FUNCTION_BLOCK TcoTixonPickVibroSeparatorTask EXTENDS TcoTixonFeedingTask
VAR_IN_OUT
	inoConfig 	: TcoTixonPickVibro_Config_v_1_x_x;
   	inoControl 	: TcoTixonPickVibro_Control_v_1_x_x;
	inoStatus 	: TcoTixonPickVibro_Status_v_1_x_x;
END_VAR
VAR
	_componentReady: BOOL;
END_VAR

IF Execute() THEN
	 
  	IF _progress = 0 THEN
		IF NOT __ISVALIDREF(inoControl) THEN
			_varInfo :=__VARINFO(inoControl);
			Messenger.Programming(_sb.Clear().Append('<#Invalid reference: #>').Append(_varInfo.Symbol).ToString()).Pin();
		ELSIF NOT __ISVALIDREF(inoConfig) THEN                                                  
			_varInfo :=__VARINFO(inoConfig);                                                    
			Messenger.Programming(_sb.Clear().Append('<#Invalid reference: #>').Append(_varInfo.Symbol).ToString()).Pin();
		ELSIF NOT __ISVALIDREF(inoStatus) THEN                                                  
			_varInfo :=__VARINFO(inoStatus);                                                    
			Messenger.Programming(_sb.Clear().Append('<#Invalid reference: #>').Append(_varInfo.Symbol).ToString()).Pin();
		ELSIF NOT inoStatus.ControllerInAuto THEN                                                  
			_varInfo :=__VARINFO(inoStatus.ControllerInAuto);                                                                                              
			Messenger.Warning(_sb.Clear().Append('<#Tixon control system not in auto #>').Append(_varInfo.Symbol).ToString());
		ELSE

			_progress := _progress + 1;

		END_IF

	END_IF
	IF _progress = 1 THEN
		inoControl.SepareComponent:=FALSE;
		_varInfo :=__VARINFO( inoStatus.SeparatorHomePos);                                                
		THIS^.Messenger.OnCondition(_infoTimer.Q AND NOT inoStatus.SeparatorHomePos).Warning(_sb.Clear().Append('<#Waiting for #>').Append(_varInfo.Symbol).ToString());
		IF  inoStatus.SeparatorHomePos THEN
			_progress := _progress + 1;
			_timer(In:=FALSE);
		END_IF;
	END_IF;
	
	
	IF _progress = 2 THEN	
		Messenger.Debug('<#Waiting for component in  separator#>');
		_timer(IN:=inoStatus.SeparatorPresent,Pt:=inoConfig.TimeToComponentInSeparator);
		IF _timer.Q THEN
			_progress := _progress + 1;
			_timer(In:=FALSE);
		END_IF
	END_IF;
	
	IF _progress = 3 THEN	
		inoControl.SepareComponent:=TRUE;
		Messenger.Debug('<#Waiting for component out of  separator#>');
		_timer(IN:=inoStatus.SeparatorPresent,Pt:=inoConfig.TimeToComponentOutSeparator);
		IF inoStatus.SeparatorPresent THEN
			_progress := _progress + 1;
			_timer(In:=FALSE);
		ELSIF _timer.Q THEN
			_progress := 1;
			_timer(In:=FALSE);
		END_IF
	END_IF;
	
	IF _progress = 4 THEN	
		_componentReady:=TRUE;
		THIS^.DoneWhen(TRUE);
	END_IF;		

   
    CallTimers(TRUE);
	
	THIS^.ThrowWhen(_errorTimer.Q );
	
END_IF

inoStatus.ComponentReady:=_componentReady;

IF  THIS^.Error AND NOT _errorMessage.Pinned THEN
	THIS^.Restore();
END_IF

PROPERTY PUBLIC ComponentReady : bool
GET
ComponentReady:=_componentReady;
END_GET
END_PROPERTY

(*~
	<docu>
		<summary>
			Executes when task is aborted.
		</summary>			
	</docu>	
~*)
METHOD PROTECTED OnAbort
IF  __ISVALIDREF(inoStatus) THEN   THIS^.inoStatus.ActionDescription := '<#Separator task  was aborted.#>'; END_IF;
END_METHOD

(*~
	<docu>
		<summary>
			Executes when task reaches the ```Done``` state .
		</summary>			
	</docu>	
~*)
METHOD PROTECTED OnDone
IF  __ISVALIDREF(inoStatus) THEN   THIS^.inoStatus.ActionDescription := '<#Separator task  finished successfully.#>'; END_IF;
_progress:=0;
IF AutoRestore THEN
	Restore();
END_IF
END_METHOD

METHOD PROTECTED OnError
VAR
	description: STRING;
END_VAR
description := '<#Separator task finished with error.#>'; 
_componentReady:=false;
IF  __ISVALIDREF(inoStatus) THEN   THIS^.inoStatus.ActionDescription := description; END_IF;
THIS^._errorMessage.Error(_sb.Clear().Append(description).Append(' To restore acknowledge this alarm.').ToString()).Pin();
END_METHOD

METHOD PROTECTED OnStart
IF  __ISVALIDREF(inoStatus) THEN  THIS^.inoStatus.ActionDescription := '<#Separator task started.#>'; END_IF; 
_componentReady:=false;
CallTimers(FALSE);
END_METHOD

(*~
	<docu>
		<summary>
			Restores this instance to the Ready state. Can be called explicitly or from within one of the restore mechanisms.
			<para>
				See also <see cref="PlcDocu.TcoCore.TcoTask.AutoRestorable()"/>
			</para>
		</summary>			
	</docu>	
~*)
METHOD Restore : ITcoRestorable
SUPER^.Restore();
_componentReady:=false;
END_METHOD

END_FUNCTION_BLOCK

(* stored: Version 1.1.0.1, ProductVersion 3.1.4024.12
   POU TcoTixonPickVibroSeparatorTask: Id {2ab41d39-2cea-0e03-0c1d-dfe7a5028895}, SpecialFunc None
   Property ComponentReady: Id {dbb351eb-4562-0100-09b4-e5af26acdf2b}
   Get Get: Id {caeab96f-fbdb-04e0-21ad-3ffc2f0b5586}
   Method OnAbort: Id {7b9c629c-fa59-0902-27cb-2dacda4eaf47}
   Method OnDone: Id {46625adb-88d2-0a7c-12d6-0c998960c653}
   Method OnError: Id {7e3a2530-2da6-0e41-07ea-0d51cec18fcb}
   Method OnStart: Id {48be983a-d0fc-0457-124c-09c0e5ca21dd}
   Method Restore: Id {e018be0b-67fd-03da-368f-cf29df911068} *)
